FUNCTION_BLOCK SFC1_VIEW (* Composite Function Block Type *)
  (* Standard: 61499-2 *)
  (* Version 0.2, 2003-12-05, JHC, Rockwell Automation, Renamed from NEWCOMPFB. *)
  (* Version 0.1, 2002-01-08, JHC, Rockwell Automation, Added DLY FB as example. *)
  (* Version 0.0, 2000-05-27, JHC, Rockwell Automation *)
  (* Compiler header: package fb.rt.pnp;import fb.rt.vhmi.*; *)
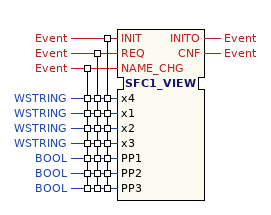
  EVENT_INPUT
    INIT WITH x4, x1, x2, x3, PP1, PP2, PP3; (* Initialization Request *)
    REQ WITH x4, x1, x2, x3, PP1, PP2, PP3; (* Normal Execution Request *)
    NAME_CHG WITH x4, x1, x2, x3, PP1, PP2, PP3;
  END_EVENT
  EVENT_OUTPUT
    INITO; (* Initialization Confirm *)
    CNF; (* Execution Confirmation *)
  END_EVENT
  VAR_INPUT
    x4 : WSTRING; (* Input event qualifier *)
    x1 : WSTRING;
    x2 : WSTRING;
    x3 : WSTRING;
    PP1 : BOOL;
    PP2 : BOOL;
    PP3 : BOOL;
  END_VAR
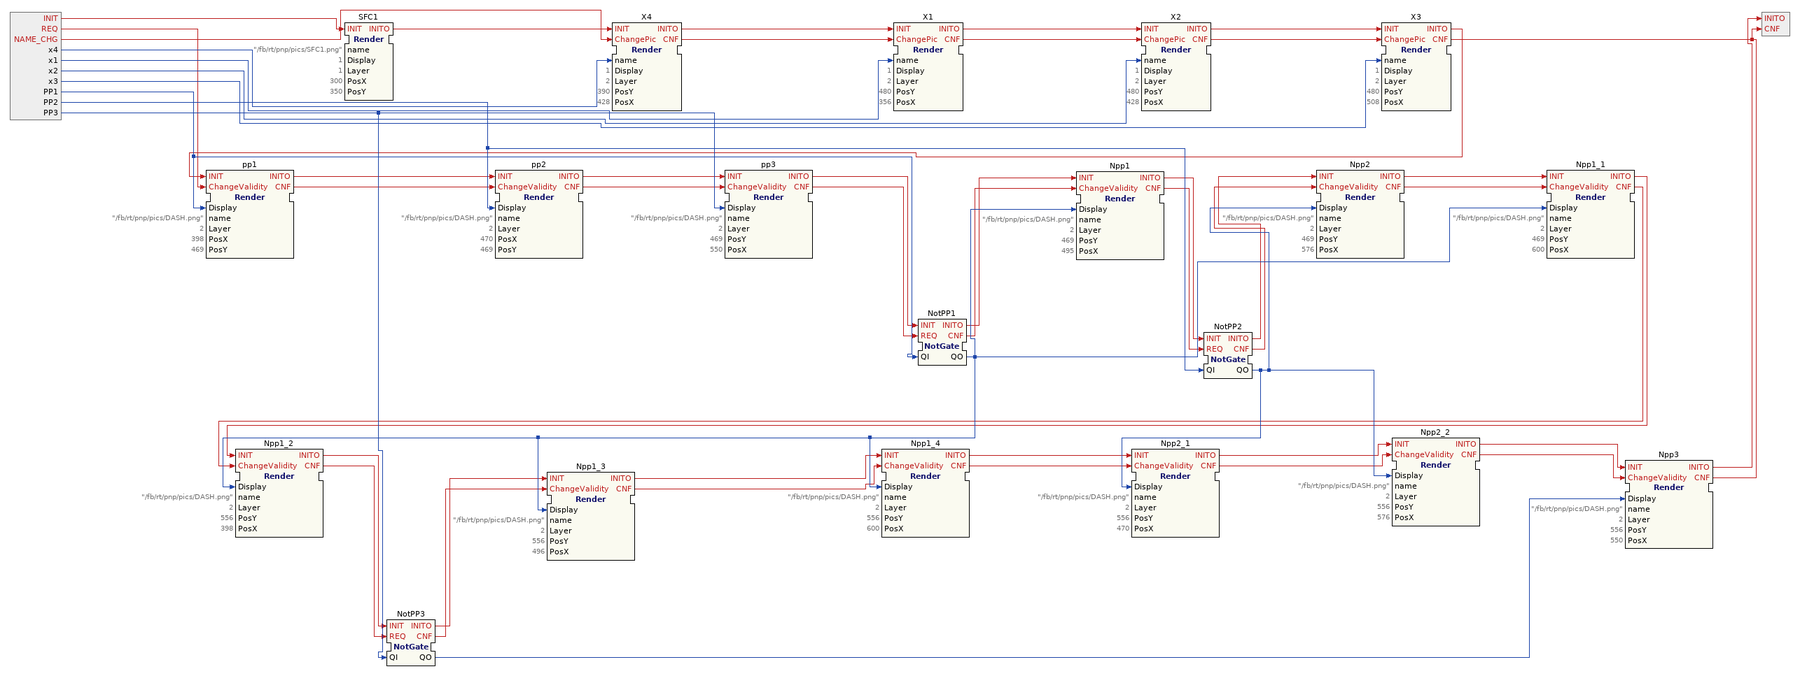
  FBS
    SFC1 : Render(name := "/fb/rt/pnp/pics/SFC1.png", Display := 1, Layer := 1, PosX := 300, PosY := 350);
    X4 : Render(Display := 1, Layer := 2, PosY := 390, PosX := 428);
    X1 : Render(Display := 1, Layer := 2, PosY := 480, PosX := 356);
    X2 : Render(Display := 1, Layer := 2, PosY := 480, PosX := 428);
    X3 : Render(Display := 1, Layer := 2, PosY := 480, PosX := 508);
    pp1 : Render(name := "/fb/rt/pnp/pics/DASH.png", Layer := 2, PosX := 398, PosY := 469);
    pp2 : Render(name := "/fb/rt/pnp/pics/DASH.png", Layer := 2, PosX := 470, PosY := 469);
    pp3 : Render(name := "/fb/rt/pnp/pics/DASH.png", Layer := 2, PosY := 469, PosX := 550);
    Npp1 : Render(name := "/fb/rt/pnp/pics/DASH.png", Layer := 2, PosY := 469, PosX := 495);
    Npp2 : Render(name := "/fb/rt/pnp/pics/DASH.png", Layer := 2, PosY := 469, PosX := 576);
    Npp1_1 : Render(name := "/fb/rt/pnp/pics/DASH.png", Layer := 2, PosY := 469, PosX := 600);
    Npp1_2 : Render(name := "/fb/rt/pnp/pics/DASH.png", Layer := 2, PosY := 556, PosX := 398);
    Npp1_3 : Render(name := "/fb/rt/pnp/pics/DASH.png", Layer := 2, PosY := 556, PosX := 496);
    Npp1_4 : Render(name := "/fb/rt/pnp/pics/DASH.png", Layer := 2, PosY := 556, PosX := 600);
    Npp2_1 : Render(name := "/fb/rt/pnp/pics/DASH.png", Layer := 2, PosY := 556, PosX := 470);
    Npp2_2 : Render(name := "/fb/rt/pnp/pics/DASH.png", Layer := 2, PosY := 556, PosX := 576);
    Npp3 : Render(name := "/fb/rt/pnp/pics/DASH.png", Layer := 2, PosY := 556, PosX := 550);
    NotPP1 : NotGate;
    NotPP2 : NotGate;
    NotPP3 : NotGate;
  END_FBS
  EVENT_CONNECTIONS
    INIT TO SFC1.INIT;
    SFC1.INITO TO X4.INIT;
    X4.INITO TO X1.INIT;
    X1.INITO TO X2.INIT;
    X2.INITO TO X3.INIT;
    X3.INITO TO pp1.INIT;
    pp1.INITO TO pp2.INIT;
    pp2.INITO TO pp3.INIT;
    Npp2.INITO TO Npp1_1.INIT;
    Npp1_1.INITO TO Npp1_2.INIT;
    Npp1_3.INITO TO Npp1_4.INIT;
    Npp1_4.INITO TO Npp2_1.INIT;
    Npp2_1.INITO TO Npp2_2.INIT;
    Npp2_2.INITO TO Npp3.INIT;
    Npp3.INITO TO INITO;
    X4.CNF TO X1.ChangePic;
    X1.CNF TO X2.ChangePic;
    X2.CNF TO X3.ChangePic;
    X3.CNF TO CNF;
    REQ TO pp1.ChangeValidity;
    pp1.CNF TO pp2.ChangeValidity;
    pp2.CNF TO pp3.ChangeValidity;
    Npp2.CNF TO Npp1_1.ChangeValidity;
    Npp1_1.CNF TO Npp1_2.ChangeValidity;
    Npp1_3.CNF TO Npp1_4.ChangeValidity;
    Npp1_4.CNF TO Npp2_1.ChangeValidity;
    Npp2_1.CNF TO Npp2_2.ChangeValidity;
    Npp2_2.CNF TO Npp3.ChangeValidity;
    Npp3.CNF TO CNF;
    pp3.INITO TO NotPP1.INIT;
    NotPP1.INITO TO Npp1.INIT;
    NotPP1.CNF TO Npp1.ChangeValidity;
    pp3.CNF TO NotPP1.REQ;
    Npp1.INITO TO NotPP2.INIT;
    NotPP2.INITO TO Npp2.INIT;
    NotPP2.CNF TO Npp2.ChangeValidity;
    Npp1.CNF TO NotPP2.REQ;
    Npp1_2.INITO TO NotPP3.INIT;
    NotPP3.INITO TO Npp1_3.INIT;
    NotPP3.CNF TO Npp1_3.ChangeValidity;
    Npp1_2.CNF TO NotPP3.REQ;
    NAME_CHG TO X4.ChangePic;
  END_CONNECTIONS
  DATA_CONNECTIONS
    PP1 TO pp1.Display;
    PP2 TO pp2.Display;
    PP3 TO pp3.Display;
    x4 TO X4.name;
    x1 TO X1.name;
    x2 TO X2.name;
    x3 TO X3.name;
    NotPP1.QO TO Npp1.Display;
    PP1 TO NotPP1.QI;
    PP2 TO NotPP2.QI;
    NotPP2.QO TO Npp2.Display;
    NotPP1.QO TO Npp1_1.Display;
    PP3 TO NotPP3.QI;
    NotPP1.QO TO Npp1_4.Display;
    NotPP2.QO TO Npp2_1.Display;
    NotPP3.QO TO Npp3.Display;
    NotPP1.QO TO Npp1_2.Display;
    NotPP1.QO TO Npp1_3.Display;
    NotPP2.QO TO Npp2_2.Display;
  END_CONNECTIONS
END_FUNCTION_BLOCK
